// TIA Portal V18 export
FUNCTION "Faults" : Void   // FC25, LAD
{ S7_Optimized_Access := 'TRUE' }
VERSION : 0.1
// stored: AutoNumber true, IsIECCheckEnabled false, SetENOAutomatically false, UDAEnableTagReadback false
   VAR_TEMP
      spare3 : Bool;
   END_VAR
BEGIN

REGION Network 1
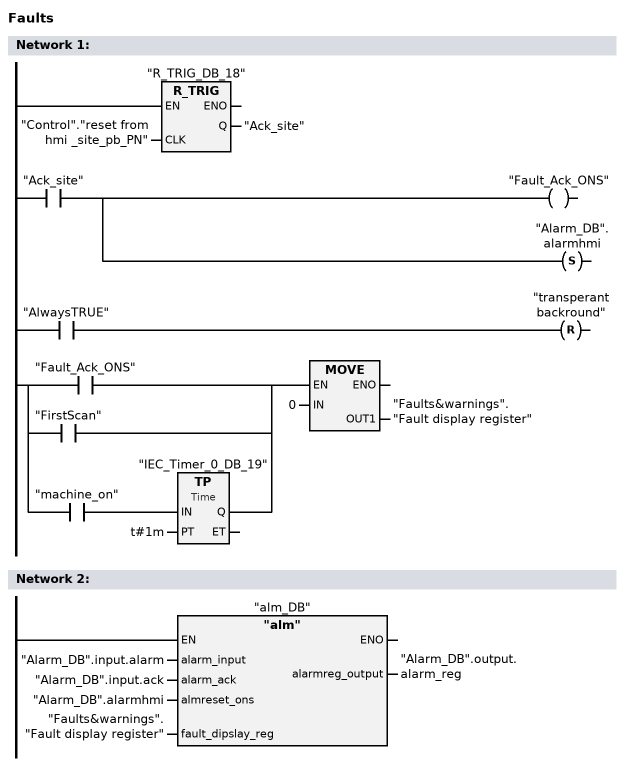
   RUNG wire#powerrail
      "R_TRIG_DB_18".R_TRIG(CLK := "Control"."reset from hmi _site_pb_PN", Q => "Ack_site")
   END_RUNG
   RUNG wire#powerrail
      Contact( "Ack_site" )
      wire#w1
      Coil( "Fault_Ack_ONS" )
   END_RUNG
   RUNG wire#w1
      S_Coil( "Alarm_DB".alarmhmi )
   END_RUNG
   RUNG wire#powerrail
      Contact( "AlwaysTRUE" )
      R_Coil( "transperant backround" )
   END_RUNG
   RUNG wire#powerrail
      Contact( "Fault_Ack_ONS" )
      wire#w2
      Move(in := 0, out1 => "Faults&warnings"."Fault display register")
   END_RUNG
   RUNG wire#powerrail
      Contact( "FirstScan" )
   END_RUNG wire#w2
   RUNG wire#powerrail
      Contact( "machine_on" )
      { S7_Templates := "time_type := Time" } "IEC_Timer_0_DB_19".TP(pt := t#1m, et =>)
   END_RUNG wire#w2
   // the same network as SCL:
   "R_TRIG_DB_18"(CLK := "Control"."reset from hmi _site_pb_PN", Q => "Ack_site");   // R_TRIG
   "Fault_Ack_ONS" := "Ack_site";
   IF "Ack_site" THEN "Alarm_DB".alarmhmi := TRUE; END_IF;
   IF "AlwaysTRUE" THEN "transperant backround" := FALSE; END_IF;
   "IEC_Timer_0_DB_19".TP(IN := "machine_on", PT := t#1m);
   IF "Fault_Ack_ONS" OR "FirstScan" OR "IEC_Timer_0_DB_19".Q THEN
       "Faults&warnings"."Fault display register" := 0;
   END_IF;
END_REGION

REGION Network 2
   RUNG wire#powerrail
      "alm_DB"(alarm_input := "Alarm_DB".input.alarm, alarm_ack := "Alarm_DB".input.ack, almreset_ons := "Alarm_DB".alarmhmi, fault_dipslay_reg := "Faults&warnings"."Fault display register", alarmreg_output => "Alarm_DB".output.alarm_reg)
   END_RUNG
   // the same network as SCL:
   "alm_DB"(alarm_input := "Alarm_DB".input.alarm,   // "alm"
            alarm_ack := "Alarm_DB".input.ack,
            almreset_ons := "Alarm_DB".alarmhmi,
            fault_dipslay_reg := "Faults&warnings"."Fault display register",
            alarmreg_output => "Alarm_DB".output.alarm_reg);
END_REGION

REGION Network 3 (SCL): Alarm FB call
   // "alm_DB"(alarm_input:=,
   //          alarmreg_output=>,
   //          alarm_ack:=,
   //          almreset_ons:=,
   //          fault_dipslay_reg:=);

   "Faults&warnings"."Fault present" := ("Faults&warnings"."Fault display register" <> 0); // fault present
   "Fault display register 1" := %DB36.;
   "Fault display register 2" := %DB36.;
   "Fault display register 3" := %DB36.;
   "Fault display register 4" := %DB36.;
   "Fault display register 5" := %DB36.;
   "Fault display register 6" := %DB36.;
END_REGION

REGION Network 4 (SCL): Alarm Register 1 ==== Fault Register 1
   "Alarm_DB".input.alarm[8] := NOT("emergency stop"); //A1-Emergenct stop active
   //"Alarm_DB".input.alarm[9] := "Faults&warnings"."Status Nok"."Drive controller A NK"; //A2-Pump A Drive Fault
   //"Alarm_DB".input.alarm[10] := "Faults&warnings"."Status Nok"."Drive controller B NK"; //A3-Pump B Drive Fault
   ////"Alarm_DB".input.alarm[11]:= agitatorA; //A4-Agitator A Fault
   ////"Alarm_DB".input.alarm[12]:= agitatorB; //A5-Agitator B Fault"
   // "Alarm_DB".input.alarm[13] := "Control".Level_sensor_enable AND ("Level Sensor A" >= 32767); //A6-Tank A level sensor fault
   // "Alarm_DB".input.alarm[14] := "Control".Level_sensor_enable AND ("Level Sensor B" >= 32767); //A7-Tank B level sensor fault
   // "Alarm_DB".input.alarm[15] := (("Control".Pressure_sensor_select = 0) AND ("Pressure sensor Pump Inlet A" >= 32767)) OR (("Control".Pressure_sensor_select = 1) AND ("Pressure sensor Pump Inlet A_mA" >= 32767));//A8-Pump A pressure sensor fault Inlet
   // "Alarm_DB".input.alarm[0] := (("Control".Pressure_sensor_select = 0) AND ("Pressure Sensor Pump Inlet B" >= 32767)) OR (("Control".Pressure_sensor_select = 1) AND ("Pressure Sensor Pump Inlet B_mA" >= 32767)); //A9-Pump B pressure sensor fault Inlet
   //"Alarm_DB".input.alarm[1] := "Re-filling Sequence DB"."Compare Re-fillingFilling sequence A"."Refilling Error";  //A10- Tank A refilling Error // not used
   //"Alarm_DB".input.alarm[2] := "Re-filling Sequence DB"."Compare Filling sequence b"."Refilling Error";  //A11- Tank B refilling Error // not used
   // "Alarm_DB".input.alarm[3] := NOT("heater status"."p100 connection okay".heater1) AND "Heater settings"."heater EN 1"; //A12-Heater1 sensor fault
   // "Alarm_DB".input.alarm[4] := NOT ("heater status"."p100 connection okay".heater2) AND "Heater settings"."heater EN 2";  //A13-Heater1 sensor fault
   // "Alarm_DB".input.alarm[5] := NOT ("heater status"."p100 connection okay".heater3) AND "Heater settings"."heater EN 3"; //A14-Heater3 sensor fault
   // "Alarm_DB".input.alarm[6] := NOT ("heater status"."p100 connection okay".heater4) AND "Heater settings"."heater EN 4";  //A15-Heater4 sensor fault
    //"Alarm_DB".input.alarm[7] := //A16-Reserve
END_REGION

REGION Network 5 (SCL): Alarm Register 2 ==== Fault Register 2
   // "Alarm_DB".input.alarm[24] := "heater status"."Limit under temperature".heater1; //"A17-Heater1 undertemperature" 
   // "Alarm_DB".input.alarm[25] := "heater status"."Limit under temperature".heater2; //A18-Heater2 undertemperature
   // "Alarm_DB".input.alarm[26] := "heater status"."Limit under temperature".heater3; //A19-Heater3 undertemperature
   // "Alarm_DB".input.alarm[27] := "heater status"."Limit under temperature".heater4; //A20-Heater4 undertemperature
   // "Alarm_DB".input.alarm[28] := "heater status"."Limit Over temperature".heater1; //"A21- Heater 1overtemperature"
   // "Alarm_DB".input.alarm[29] := "heater status"."Limit Over temperature".heater2; //"A22- Heater2 overtemperature"
   // "Alarm_DB".input.alarm[30] := "heater status"."Limit Over temperature".heater3; //"A23- Heater3 overtemperature"
   // "Alarm_DB".input.alarm[31] := "heater status"."Limit Over temperature".heater4; //"A24- Heater4 overtemperature"
    //"Alarm_DB".input.alarm[16] := //A25- Reserve
    //"Alarm_DB".input.alarm[17] := //A26- Reserve
    //"Alarm_DB".input.alarm[18] := //A27- Reserve
   // "Alarm_DB".input.alarm[19] := "Faults&warnings"."Status Nok"."Over pressure A inlet"; //A28- Pump A Inlet over pressure
   // "Alarm_DB".input.alarm[20] := "Faults&warnings"."Status Nok"."Over pressure B inlet"; //A29- Pump B Inlet over pressure
   // "Alarm_DB".input.alarm[21] := "Faults&warnings"."Status Nok"."Level empty A1" OR "Temp".bit20 ; //A30-Tank A1 Level Empty
   // //"Alarm_DB".input.alarm[22] := //A31-Reserve
   // "Alarm_DB".input.alarm[23] := "Faults&warnings"."Status Nok"."Level empty B1" OR "Temp".bit21; //A32-Tank B Level Empty
END_REGION

REGION Network 6 (SCL): Alarm Register 3 ==== Fault Register 3
   // "Alarm_DB".input.alarm[40] := "Faults&warnings"."Status Nok"."Low level A1"; //A33-Tank A1 low level 
   // //"Alarm_DB".input.alarm[41] :=  //A34-Reserve
   // "Alarm_DB".input.alarm[42] := "Faults&warnings"."Status Nok"."Low level B1"; //A35-Tank B low level
   // "Alarm_DB".input.alarm[43] := "pressure"."Control A"."under pressure Occured"; //A36-Pump A Inlet lower pressure
   // "Alarm_DB".input.alarm[44] := "pressure"."Control B"."under pressure Occured"; //A37-Pump B Inlet lower pressure
   // //"Alarm_DB".input.alarm[45] :=  //A38-Reserve
   // //"Alarm_DB".input.alarm[46] :=  //A39-Reserve
   "Alarm_DB".input.alarm[47] := "Potlife".contol."Potlife elapsed machine not in regeneration" AND NOT ("Functions"."2k"."pre run program selected") AND NOT ("Metering".Metering_running);  //A40-Potlife elapsed Change static mixer
    //"Alarm_DB".input.alarm[32] := //A41-Reserve
    //"Alarm_DB".input.alarm[33] := //A42-Reserve
    //"Alarm_DB".input.alarm[34] := //A43-Reserve
    //"Alarm_DB".input.alarm[35] := //A44-Reserve
    //"Alarm_DB".input.alarm[36] := //A45-Reserve
    //"Alarm_DB".input.alarm[37] := //A46-Reserve
   //"Alarm_DB".input.alarm[38] := //A47-Reserve
   //"Alarm_DB".input.alarm[39] := //A48-Reserve
END_REGION

REGION Network 7 (SCL): Alarm Register 4 ==== Fault Register 4
   //"Alarm_DB".input.alarm[56] :=  //A49-Reserve
   //"Alarm_DB".input.alarm[57] :=  //A50-Reserve
   //"Alarm_DB".input.alarm[58] := ///A51-Reserve
   //"Alarm_DB".input.alarm[59] := //A52-Reserve
   //"Alarm_DB".input.alarm[60] := //A53-Reserve
   //"Alarm_DB".input.alarm[61] :=  //A54-Reserve
   //"Alarm_DB".input.alarm[62] :=  //A55-Reserve
   //"Alarm_DB".input.alarm[63] := //A56-Reserve
    //"Alarm_DB".input.alarm[48] := //A57-Reserve
    //"Alarm_DB".input.alarm[49] := //A58-Reserve
    //"Alarm_DB".input.alarm[50] := //A59-Reserve
    //"Alarm_DB".input.alarm[51] := //A60-Reserve
    //"Alarm_DB".input.alarm[52] := //A61-Reserve
    //"Alarm_DB".input.alarm[53] := "Faults&warnings"."Status Nok"."Flowrate error"; //A62-Reserve
   //"Alarm_DB".input.alarm[54] := //A63-Reserve
   //"Alarm_DB".input.alarm[55] := //A64-Reserve
END_REGION

REGION Network 8 (SCL): Alarm Register 5 ==== Fault Register 5
   //"Alarm_DB".input.alarm[72] :=  //A65-Reserve
   //"Alarm_DB".input.alarm[73] :=  //A66-Reserve
   //"Alarm_DB".input.alarm[74] := ///A67-Reserve
   //"Alarm_DB".input.alarm[75] := //A68-Reserve
   //"Alarm_DB".input.alarm[76] := //A69-Reserve
   //"Alarm_DB".input.alarm[77] := "Mixing ratio"."mixing ratio Low Warning"; //A70-Warning mixing ratio low
   //"Alarm_DB".input.alarm[78] := "Mixing ratio"."mixing ratio high Warning"; //A71- warning Mixing Ratio high
   //"Alarm_DB".input.alarm[79] := "Mixing ratio"."Mixing ratio Low  Error"; //A72- Error Mixing ratio Low
   //"Alarm_DB".input.alarm[64] := "Mixing ratio"."Mixing ratio high Error"; //A73- Error Mixing Ratio high
    //"Alarm_DB".input.alarm[65] := //A74-Reserve
    //"Alarm_DB".input.alarm[66] := //A75-Reserve
    //"Alarm_DB".input.alarm[67] := //A76-Reserve
    //"Alarm_DB".input.alarm[68] := //A77-Reserve
    //"Alarm_DB".input.alarm[69] := //A78-Reserve
   //"Alarm_DB".input.alarm[70] := //A79-Reserve
   //"Alarm_DB".input.alarm[71] := //A80-Reserve
END_REGION

REGION Network 9 (SCL): Alarm Register 6 ==== Fault Register 6
   // //"Alarm_DB".input.alarm[88] := //A81-Reserve
   // "Alarm_DB".input.alarm[89] := "level"."Drum Level Low A1"; //"A82-Level Low Drum A1"
   // "Alarm_DB".input.alarm[90] := "level"."Drum Level Low B1"; //"A83-Level Low Drum B1"
   // "Alarm_DB".input.alarm[91] := "level"."Drum Level Low A2"; //"A84-Level Low Drum A2"
   // "Alarm_DB".input.alarm[92] := "level"."Drum Level Low B2"; //"A85-Level Low Drum B2"
   // "Alarm_DB".input.alarm[93] := "level"."Drum Level Empty A1"; //"A86-Level Empty Drum A1"
   // "Alarm_DB".input.alarm[94] := "level"."Drum Level Empty B1";//"A87-Level Empty Drum B1"
   // "Alarm_DB".input.alarm[95] := "level"."Drum Level Empty A2"; //"A88-Level Empty Drum A2"
   // "Alarm_DB".input.alarm[80] := "level"."Drum Level Empty B2"; //"A89-Level Empty Drum B2"
   // "Temp".bit20 := ("HMI".supplySelection = 1) AND "level"."Drum Level Empty A1" AND "level"."Drum Level Empty A2";
   // "Temp".bit21 := ("HMI".supplySelection = 1) AND "level"."Drum Level Empty B1" AND "level"."Drum Level Empty B2";
   // "Alarm_DB".input.alarm[81] := "Faults&warnings"."Status Nok"."Pressure sensor Pump A Outlet"; //"A90 Pressure sensor Pump A Outlet Fault"
   // "Alarm_DB".input.alarm[82] := "Faults&warnings"."Status Nok"."Pressure Sensor Pump B Outlet"; //"A91 Pressure sensor Pump B Outlet Fault"
   // "Alarm_DB".input.alarm[83] := "Faults&warnings"."Status Nok"."Over pressure A outlet"; //A92- Pump A Outlet Over PRessure
   // "Alarm_DB".input.alarm[84] := "Faults&warnings"."Status Nok"."Over pressure B outlet"; //"A93 Over pressure B outlet"
   // "Alarm_DB".input.alarm[85] := "pressure"."Control A_Outlet"."under pressure Occured"; //A94- Pump A Outlet Under Pressure
   // "Alarm_DB".input.alarm[86] := "pressure"."Control B_Outlet"."under pressure Occured"; //"A95- Pump B Outlet Under Pressure"
   // //"Alarm_DB".input.alarm[87] := //A96-Reserve
END_REGION
END_FUNCTION
